INTERFACE I_OutputPortChangedEvent extends I_Event

PROPERTY PUBLIC Target : I_OutputPort
GET
END_GET
END_PROPERTY

END_INTERFACE

(* stored: Version 1.1.0.1, ProductVersion 3.1.4024.12
   Itf I_OutputPortChangedEvent: Id {36dbc39b-80b2-4b77-a0c7-465592c7363a}
   Property Target: Id {c45bdc57-5eac-41ac-83cd-339cce8a09ac}
   Get Get: Id {7e49caf3-05e0-40cb-94ac-218dc054eae1} *)
